TYPE stTarget :
STRUCT
	name : STRING(80);
	frameId : INT;
END_STRUCT
END_TYPE

(* stored: Version 1.1.0.1, ProductVersion 3.1.4026.18
   DUT stTarget: Id {c1b2c3d4-2222-2222-2222-222222222222} *)
